{attribute 'qualified_only'}
{attribute 'strict'}
TYPE E_Cylinder :
(
	enum_member := 0
);
END_TYPE

(* stored: Version 1.1.0.1, ProductVersion 3.1.4024.12
   DUT E_Cylinder: Id {fef6d8ca-d0ad-4a70-a1fa-f5275c29ebc1} *)
